// TIA Portal V20 export
DATA_BLOCK "OneMES_ControlData"   // DB20230
{ S7_Optimized_Access := 'TRUE' }
// stored: AutoNumber false, MemoryReserve 100
   VAR
      HMI { S7_SetPoint := 'True'} : "UDT_OneMES_HMI_Control";
      MsgDisplay { S7_SetPoint := 'True'} : "UDT_MesMsgDisplay";
      Pluse { S7_SetPoint := 'True'} : Array[0..7] of Bool;
      OP : Array[1.."OP_Sum"] of "UDT_MESControl";
   END_VAR
BEGIN
   HMI.OP_Select := 1;
   HMI.PageCount := 1;
   // MsgDisplay.OP_Sel : 工站选择/暂不使用
   OP[1]."Timer"[1..15].PT := T#1s;
END_DATA_BLOCK
